// TIA Portal project "故障读取测试" (V16)

(* hardware
DEVICE "S7-1200 station_1"  S7-1200 Station
   slot 0: "Rack_0"  S7-1200 Rack  Rack  V1.0
   slot 1: "PLC_1"  CPU 1214C DC/DC/DC  6ES7 214-1AG40-0XB0  V4.4
*)

// ===== PLC "PLC_1"  CPU 1214C DC/DC/DC =====

VAR_GLOBAL   // PLC tag table "默认变量表"
   "System_Byte" AT %MB1 : Byte;
   "FirstScan" AT %M1.0 : Bool;
   "DiagStatusUpdate" AT %M1.1 : Bool;
   "AlwaysTRUE" AT %M1.2 : Bool;
   "AlwaysFALSE" AT %M1.3 : Bool;
   "Clock_Byte" AT %MB0 : Byte;
   "Clock_10Hz" AT %M0.0 : Bool;
   "Clock_5Hz" AT %M0.1 : Bool;
   "Clock_2.5Hz" AT %M0.2 : Bool;
   "Clock_2Hz" AT %M0.3 : Bool;
   "Clock_1.25Hz" AT %M0.4 : Bool;
   "Clock_1Hz" AT %M0.5 : Bool;
   "Clock_0.625Hz" AT %M0.6 : Bool;
   "Clock_0.5Hz" AT %M0.7 : Bool;
END_VAR

DATA_BLOCK "数据块_1"   // DB3000
{ S7_Optimized_Access := 'FALSE' }
VERSION : 0.1
   VAR
      Alarm : Array[0..15] of Bool;
   END_VAR
BEGIN
   // Alarm[0] : A
   // Alarm[1] : B
   // Alarm[2] : W
   // Alarm[3] : W
   // Alarm[4] : EE
   // Alarm[5] : 6
   // Alarm[6] : 7
   // Alarm[7] : 8
   // Alarm[8] : R
   // Alarm[9] : Y
   // Alarm[10] : T
   // Alarm[11] : 12
   // Alarm[12] : 13
   // Alarm[13] : 14
   // Alarm[14] : 15
   // Alarm[15] : 16
END_DATA_BLOCK

DATA_BLOCK "数据块_2"   // DB3001
{ S7_Optimized_Access := 'FALSE' }
VERSION : 0.1
   VAR
      Alarm : Array[0..15] of Bool;
   END_VAR
BEGIN
   // Alarm[0] : 1
   // Alarm[1] : 2
   // Alarm[2] : 3
   // Alarm[3] : 4
   // Alarm[4] : 5
   // Alarm[5] : 6
   // Alarm[6] : 7
   // Alarm[7] : 8
   // Alarm[8] : 9
   // Alarm[9] : 10
   // Alarm[10] : 11
   // Alarm[11] : 12
   // Alarm[12] : 13
   // Alarm[13] : 14
   // Alarm[14] : 15
   // Alarm[15] : 16
END_DATA_BLOCK

ORGANIZATION_BLOCK "Main"   // OB1, LAD, ProgramCycle
TITLE = "Main Program Sweep (Cycle)"
{ S7_Optimized_Access := 'TRUE' }
VERSION : 0.1
   VAR_INPUT
      Initial_Call : Bool;   // Initial call of this OB
      Remanence : Bool;   // =True, if remanent data are available
   END_VAR
BEGIN
END_ORGANIZATION_BLOCK